// TIA Portal V15.1 export
// export: Created 2024-06-21T08:41:07.9526464Z, ExportSetting WithDefaults, DisplayName Totally Integrated Automation Portal, DisplayVersion V15.1 Update 5, DisplayName TIA Portal Openness, DisplayVersion V15.1 Update 5, DisplayName SINAMICS Startdrive Advanced, DisplayVersion V15.1, DisplayName G130, G150, S120, S150, SINAMICS MV, S210, DisplayVersion V15.1, DisplayName G110M, G120, G120C, G120D, G120P, DisplayVersion V15.1, DisplayName STEP 7 Professional, DisplayVersion V15.1 Update 5, DisplayName STEP 7 Safety, DisplayVersion V15.1, DisplayName WinCC Professional, DisplayVersion V15.1 Update 5, DisplayName SIMATIC Visualization Architect, DisplayVersion V15.1
FUNCTION_BLOCK "LGBInfeedOutfeed"   // FB6694, FBD
TITLE = LGBInfeedOutfeed
{ S7_Optimized_Access := 'TRUE' }
VERSION : 0.1
// stored: AutoNumber false, IsIECCheckEnabled false, IsRetainMemResEnabled false, MemoryReserve 100, SetENOAutomatically False, UDAEnableTagReadback false
   VAR_INPUT
      I_SelSwInfeed { ExternalAccessible := 'False'; ExternalVisible := 'False'; ExternalWritable := 'False'} : Bool;   // Selection switch Infeed selected
      I_SelSwOutfeed { ExternalAccessible := 'False'; ExternalVisible := 'False'; ExternalWritable := 'False'} : Bool;   // Selection switch Outfeed selected
      I_PBAcknowledge { ExternalAccessible := 'False'; ExternalVisible := 'False'; ExternalWritable := 'False'} : Bool;   // Pushbutton Acknowledge
      I_Pedal { ExternalAccessible := 'False'; ExternalVisible := 'False'; ExternalWritable := 'False'} : Bool;   // Pedal
      I_StopDet { ExternalAccessible := 'False'; ExternalVisible := 'False'; ExternalWritable := 'False'} : Bool;   // Stop detection roller during infeed
      I_ExtOutfeedReq { ExternalAccessible := 'False'; ExternalVisible := 'False'; ExternalWritable := 'False'} : Bool;   // External Outfeed request
      I_TrfOutRdyRcv { ExternalAccessible := 'False'; ExternalVisible := 'False'; ExternalWritable := 'False'} : Bool;   // Ready to Receive: Signal from next object
      I_TrfOutArrived { ExternalAccessible := 'False'; ExternalVisible := 'False'; ExternalWritable := 'False'} : Bool;   // Body Arrived: Signal from next object
      I_TrfInRdyDlv { ExternalAccessible := 'False'; ExternalVisible := 'False'; ExternalWritable := 'False'} : Bool;   // Ready to deliver: Signal from previous object
      I_TrfInTM { ExternalAccessible := 'False'; ExternalVisible := 'False'; ExternalWritable := 'False'} : Bool;   // Transfer busy signal from previous equipement
      C_TimeNotStopDet { ExternalAccessible := 'False'; ExternalVisible := 'False'; ExternalWritable := 'False'} : DInt;   // Time value for handshake signal "Arrived" by Infeed
   END_VAR
   VAR_OUTPUT
      O_TrfOutRdyDlv { ExternalAccessible := 'False'; ExternalVisible := 'False'; ExternalWritable := 'False'} : Bool;   // Ready to Deliver: Signal to next object
      O_TrfOutTM { ExternalAccessible := 'False'; ExternalVisible := 'False'; ExternalWritable := 'False'} : Bool;   // Transfer: Signal to next object
      O_TrfInRdyRcv { ExternalAccessible := 'False'; ExternalVisible := 'False'; ExternalWritable := 'False'} : Bool;   // Ready to Receive: Signal to previous object
      O_TrfInArrived { ExternalAccessible := 'False'; ExternalVisible := 'False'; ExternalWritable := 'False'} : Bool;   // Body Arrived: Signal to previous object
      O_ReqInfeed { ExternalAccessible := 'False'; ExternalVisible := 'False'; ExternalWritable := 'False'} : Bool;   // Infeed request / Led Infeed/Outfeed
      O_ReqOutfeed { ExternalAccessible := 'False'; ExternalVisible := 'False'; ExternalWritable := 'False'} : Bool;   // Outfeed request / Led Infeed/Outfeed
      O_LedInfeedOutfeed { ExternalAccessible := 'False'; ExternalVisible := 'False'; ExternalWritable := 'False'} : Bool;   // Led Infeed/Outfeed
      O_LedAcknowledge { ExternalAccessible := 'False'; ExternalVisible := 'False'; ExternalWritable := 'False'} : Bool;   // Led Acknowledge
      O_AlarmABCondition { ExternalAccessible := 'False'; ExternalVisible := 'False'; ExternalWritable := 'False'} : Bool;   // Alarm AB Condition
      O_AlarmA { ExternalAccessible := 'False'; ExternalVisible := 'False'; ExternalWritable := 'False'} : Bool;   // Alarm A
      O_AlarmB { ExternalAccessible := 'False'; ExternalVisible := 'False'; ExternalWritable := 'False'} : Bool;   // Alarm B
      O_AlarmC { ExternalAccessible := 'False'; ExternalVisible := 'False'; ExternalWritable := 'False'} : Bool;   // Alarm C
      O_AlarmD { ExternalAccessible := 'False'; ExternalVisible := 'False'; ExternalWritable := 'False'} : Bool;   // Alarm D
      H_AlarmDWord { ExternalAccessible := 'False'; ExternalVisible := 'False'; ExternalWritable := 'False'} : DWord;   // HMI Animation
   END_VAR
   VAR_IN_OUT
      IO_Modes : "Modes";   // Modes
      H_HMI : "H_HMI";   // Animation
      H_GBInfeedOutfeed : "H_GBInfeedOutfeed";   // Animation
   END_VAR
   VAR
      TrfOutRdyDlv { ExternalAccessible := 'False'; ExternalVisible := 'False'; ExternalWritable := 'False'} : Bool;   // Ready to Deliver: Signal to next object
      TrfOutTM { ExternalAccessible := 'False'; ExternalVisible := 'False'; ExternalWritable := 'False'} : Bool;   // Transfer: Signal to next object
      TrfInRdyRcv { ExternalAccessible := 'False'; ExternalVisible := 'False'; ExternalWritable := 'False'} : Bool;   // Ready to Receive: Signal to previous object
      TrfInArrived { ExternalAccessible := 'False'; ExternalVisible := 'False'; ExternalWritable := 'False'} : Bool;   // Body Arrived: Signal to previous object
      InfeedSel { ExternalAccessible := 'False'; ExternalVisible := 'False'; ExternalWritable := 'False'} : Bool;   // Infeed selected
      OutfeedSel { ExternalAccessible := 'False'; ExternalVisible := 'False'; ExternalWritable := 'False'} : Bool;   // Outfeed selected
      NotStopDetDelayed { ExternalAccessible := 'False'; ExternalVisible := 'False'; ExternalWritable := 'False'} : Bool;   // Not Stop detection delayted
      LedFeedInFeedOut { ExternalAccessible := 'False'; ExternalVisible := 'False'; ExternalWritable := 'False'} : Bool;   // Led Infeed/Outfeed
      LedAcknowledge { ExternalAccessible := 'False'; ExternalVisible := 'False'; ExternalWritable := 'False'} : Bool;   // Led Acknowledge
      ActNotStopDetDelayed { ExternalAccessible := 'False'; ExternalVisible := 'False'; ExternalWritable := 'False'} : DInt;   // Actual time Not Stop detection delayted
      AlarmA { ExternalAccessible := 'False'; ExternalVisible := 'False'; ExternalWritable := 'False'} : Bool;   // Alarm A
      AlarmB { ExternalAccessible := 'False'; ExternalVisible := 'False'; ExternalWritable := 'False'} : Bool;   // Alarm B
      AlarmC { ExternalAccessible := 'False'; ExternalVisible := 'False'; ExternalWritable := 'False'} : Bool;   // Alarm C
      AlarmD { ExternalAccessible := 'False'; ExternalVisible := 'False'; ExternalWritable := 'False'} : Bool;   // Alarm D
      AlarmABCondition { ExternalAccessible := 'False'; ExternalVisible := 'False'; ExternalWritable := 'False'} : Bool;   // Alarm AB Condition
      TimerNotStopDetDelayed { ExternalAccessible := 'False'; ExternalVisible := 'False'; ExternalWritable := 'False'} : "LTimer";   // FB
   END_VAR
   VAR_TEMP   // added for the SCL form of the ladder/FBD networks
      _w1 : Bool;
   END_VAR
BEGIN

REGION Network 1: **** 4.3 - Machine status - Operator selections **** Infeed selected
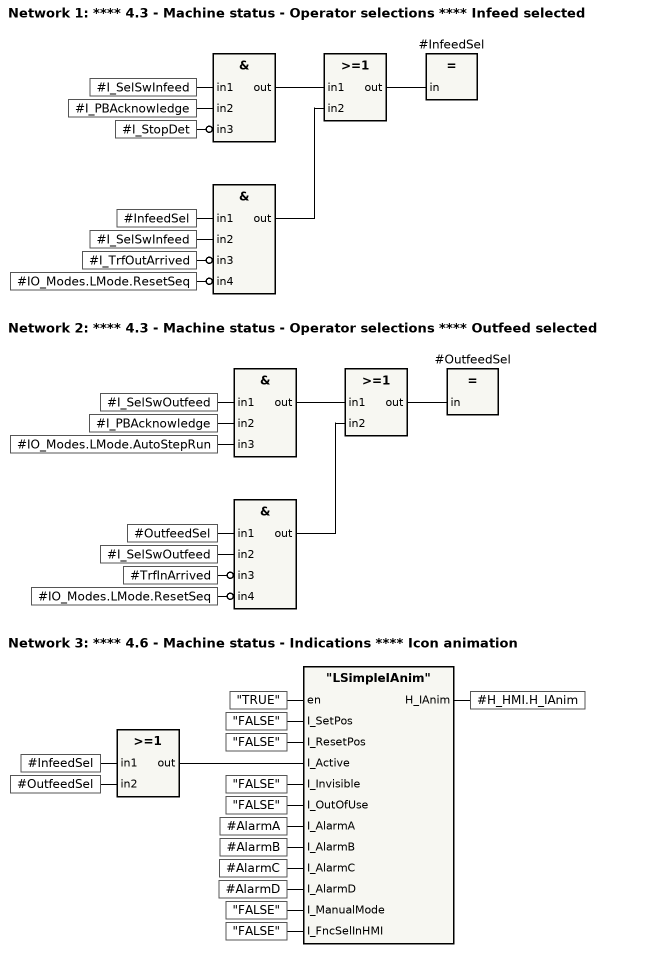
   #InfeedSel := (#I_SelSwInfeed AND #I_PBAcknowledge AND NOT #I_StopDet) OR (#InfeedSel AND #I_SelSwInfeed AND NOT #I_TrfOutArrived AND NOT #IO_Modes.LMode.ResetSeq);
END_REGION

REGION Network 2: **** 4.3 - Machine status - Operator selections **** Outfeed selected
   #OutfeedSel := (#I_SelSwOutfeed AND #I_PBAcknowledge AND #IO_Modes.LMode.AutoStepRun) OR (#OutfeedSel AND #I_SelSwOutfeed AND NOT #TrfInArrived AND NOT #IO_Modes.LMode.ResetSeq);
END_REGION

REGION Network 3: **** 4.6 - Machine status - Indications **** Icon animation
   // Icon animation
   IF "TRUE" THEN
       "LSimpleIAnim"(I_SetPos := "FALSE",
                      I_ResetPos := "FALSE",
                      I_Active := #InfeedSel OR #OutfeedSel,
                      I_Invisible := "FALSE",
                      I_OutOfUse := "FALSE",
                      I_AlarmA := #AlarmA,
                      I_AlarmB := #AlarmB,
                      I_AlarmC := #AlarmC,
                      I_AlarmD := #AlarmD,
                      I_ManualMode := "FALSE",
                      I_FncSelInHMI := "FALSE",
                      H_IAnim => #H_HMI.H_IAnim);
   END_IF;
END_REGION

REGION Network 4: **** 4.6 - Machine status - Indications **** Animation
   // Animation
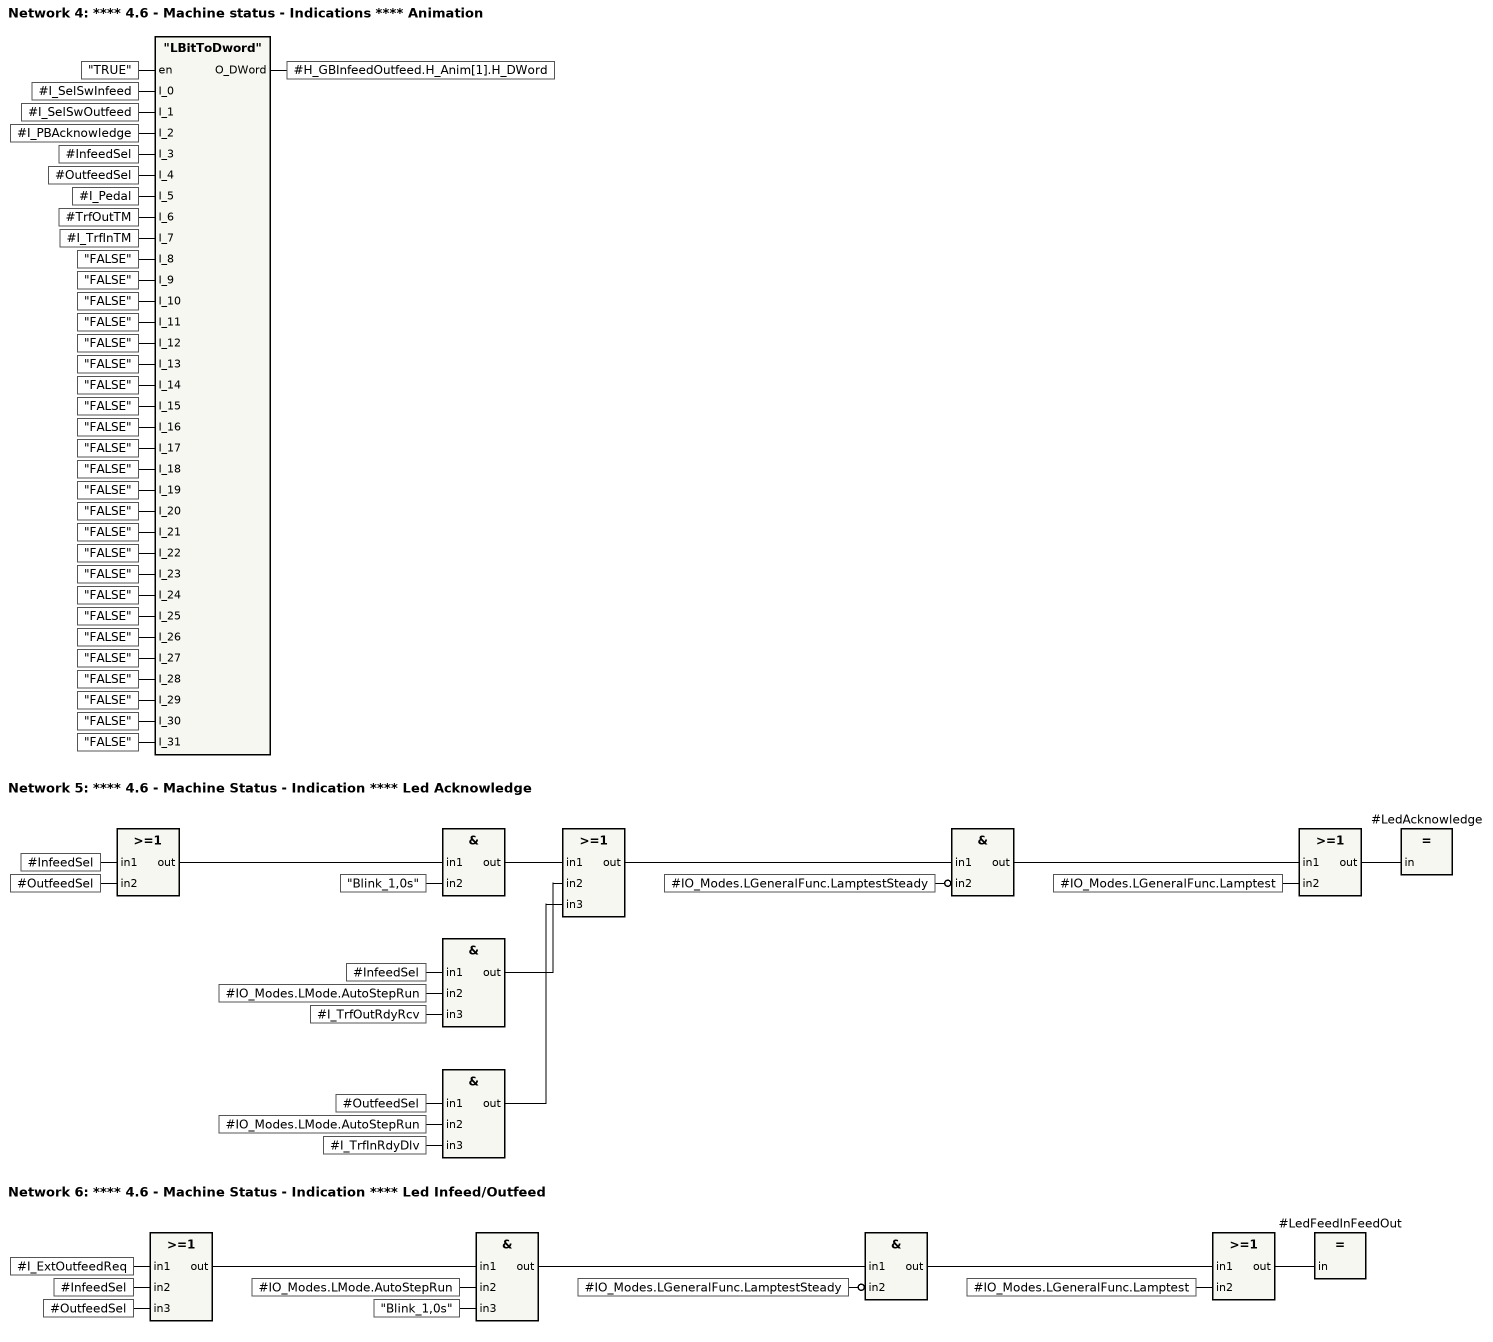
   IF "TRUE" THEN
       "LBitToDword"(I_0 := #I_SelSwInfeed,
                     I_1 := #I_SelSwOutfeed,
                     I_2 := #I_PBAcknowledge,
                     I_3 := #InfeedSel,
                     I_4 := #OutfeedSel,
                     I_5 := #I_Pedal,
                     I_6 := #TrfOutTM,
                     I_7 := #I_TrfInTM,
                     I_8 := "FALSE",
                     I_9 := "FALSE",
                     I_10 := "FALSE",
                     I_11 := "FALSE",
                     I_12 := "FALSE",
                     I_13 := "FALSE",
                     I_14 := "FALSE",
                     I_15 := "FALSE",
                     I_16 := "FALSE",
                     I_17 := "FALSE",
                     I_18 := "FALSE",
                     I_19 := "FALSE",
                     I_20 := "FALSE",
                     I_21 := "FALSE",
                     I_22 := "FALSE",
                     I_23 := "FALSE",
                     I_24 := "FALSE",
                     I_25 := "FALSE",
                     I_26 := "FALSE",
                     I_27 := "FALSE",
                     I_28 := "FALSE",
                     I_29 := "FALSE",
                     I_30 := "FALSE",
                     I_31 := "FALSE",
                     O_DWord => #H_GBInfeedOutfeed.H_Anim[1].H_DWord);
   END_IF;
END_REGION

REGION Network 5: **** 4.6 - Machine Status - Indication **** Led Acknowledge
   #LedAcknowledge := ((((#InfeedSel OR #OutfeedSel) AND "Blink_1,0s") OR (#InfeedSel AND #IO_Modes.LMode.AutoStepRun AND #I_TrfOutRdyRcv) OR (#OutfeedSel AND #IO_Modes.LMode.AutoStepRun AND #I_TrfInRdyDlv)) AND NOT #IO_Modes.LGeneralFunc.LamptestSteady) OR #IO_Modes.LGeneralFunc.Lamptest;
END_REGION

REGION Network 6: **** 4.6 - Machine Status - Indication **** Led Infeed/Outfeed
   #LedFeedInFeedOut := ((#I_ExtOutfeedReq OR #InfeedSel OR #OutfeedSel) AND #IO_Modes.LMode.AutoStepRun AND "Blink_1,0s" AND NOT #IO_Modes.LGeneralFunc.LamptestSteady) OR #IO_Modes.LGeneralFunc.Lamptest;
END_REGION

REGION Network 7: **** 5.2 - Equations - Flow Equation **** Timer Not StopDet Delayed
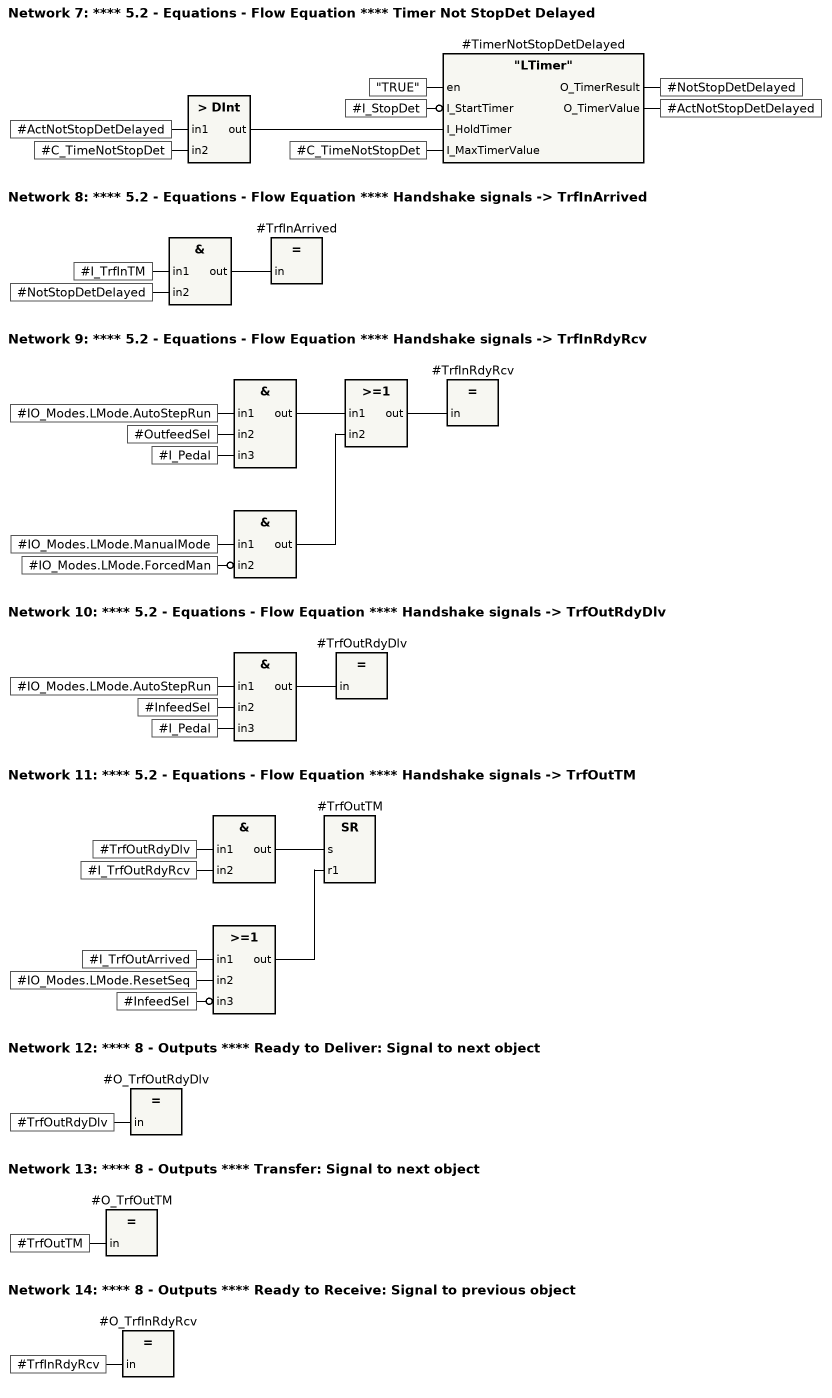
   IF "TRUE" THEN
       #TimerNotStopDetDelayed(I_StartTimer := NOT #I_StopDet,   // "LTimer"
                               I_HoldTimer := #ActNotStopDetDelayed > #C_TimeNotStopDet,
                               I_MaxTimerValue := #C_TimeNotStopDet,
                               O_TimerResult => #NotStopDetDelayed,
                               O_TimerValue => #ActNotStopDetDelayed);
   END_IF;
END_REGION

REGION Network 8: **** 5.2 - Equations - Flow Equation **** Handshake signals -> TrfInArrived
   #TrfInArrived := #I_TrfInTM AND #NotStopDetDelayed;
END_REGION

REGION Network 9: **** 5.2 - Equations - Flow Equation **** Handshake signals -> TrfInRdyRcv
   #TrfInRdyRcv := (#IO_Modes.LMode.AutoStepRun AND #OutfeedSel AND #I_Pedal) OR (#IO_Modes.LMode.ManualMode AND NOT #IO_Modes.LMode.ForcedMan);
END_REGION

REGION Network 10: **** 5.2 - Equations - Flow Equation **** Handshake signals -> TrfOutRdyDlv
   #TrfOutRdyDlv := #IO_Modes.LMode.AutoStepRun AND #InfeedSel AND #I_Pedal;
END_REGION

REGION Network 11: **** 5.2 - Equations - Flow Equation **** Handshake signals -> TrfOutTM
   IF #TrfOutRdyDlv AND #I_TrfOutRdyRcv THEN
       #TrfOutTM := TRUE;   // SR flip-flop
   END_IF;
   IF #I_TrfOutArrived OR #IO_Modes.LMode.ResetSeq OR NOT #InfeedSel THEN #TrfOutTM := FALSE; END_IF;
END_REGION

REGION Network 12: **** 8 - Outputs **** Ready to Deliver: Signal to next object
   #O_TrfOutRdyDlv := #TrfOutRdyDlv;
END_REGION

REGION Network 13: **** 8 - Outputs **** Transfer: Signal to next object
   #O_TrfOutTM := #TrfOutTM;
END_REGION

REGION Network 14: **** 8 - Outputs **** Ready to Receive: Signal to previous object
   #O_TrfInRdyRcv := #TrfInRdyRcv;
END_REGION

REGION Network 15: **** 8 - Outputs **** Body Arrived: Signal to previous object
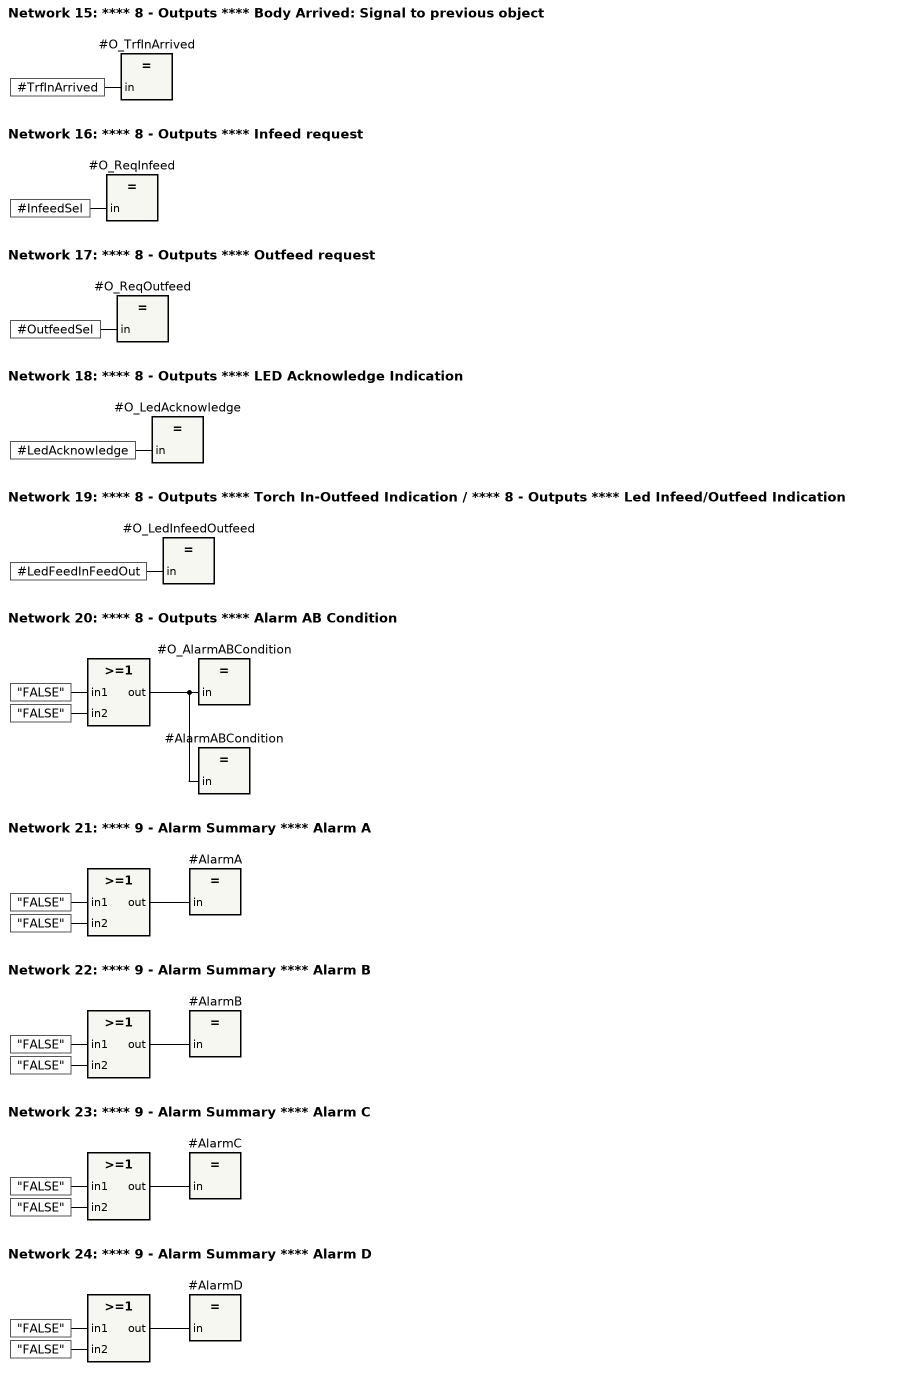
   #O_TrfInArrived := #TrfInArrived;
END_REGION

REGION Network 16: **** 8 - Outputs **** Infeed request
   #O_ReqInfeed := #InfeedSel;
END_REGION

REGION Network 17: **** 8 - Outputs **** Outfeed request
   #O_ReqOutfeed := #OutfeedSel;
END_REGION

REGION Network 18: **** 8 - Outputs **** LED Acknowledge Indication
   #O_LedAcknowledge := #LedAcknowledge;
END_REGION

REGION Network 19: **** 8 - Outputs **** Torch In-Outfeed Indication / **** 8 - Outputs **** Led Infeed/Outfeed Indication
   #O_LedInfeedOutfeed := #LedFeedInFeedOut;
END_REGION

REGION Network 20: **** 8 - Outputs **** Alarm AB Condition
   // Alarm AB Condition
   #O_AlarmABCondition := "FALSE" OR "FALSE";
   #AlarmABCondition := #O_AlarmABCondition;
END_REGION

REGION Network 21: **** 9 - Alarm Summary **** Alarm A
   // Alarm A
   #AlarmA := "FALSE" OR "FALSE";
END_REGION

REGION Network 22: **** 9 - Alarm Summary **** Alarm B
   // Alarm B
   #AlarmB := "FALSE" OR "FALSE";
END_REGION

REGION Network 23: **** 9 - Alarm Summary **** Alarm C
   // Alarm C
   #AlarmC := "FALSE" OR "FALSE";
END_REGION

REGION Network 24: **** 9 - Alarm Summary **** Alarm D
   // Alarm D
   #AlarmD := "FALSE" OR "FALSE";
END_REGION

REGION Network 25: **** 9 - Alarm Summary **** Alarms To Alarm UDT Alarms To Alarm UDT Get Name
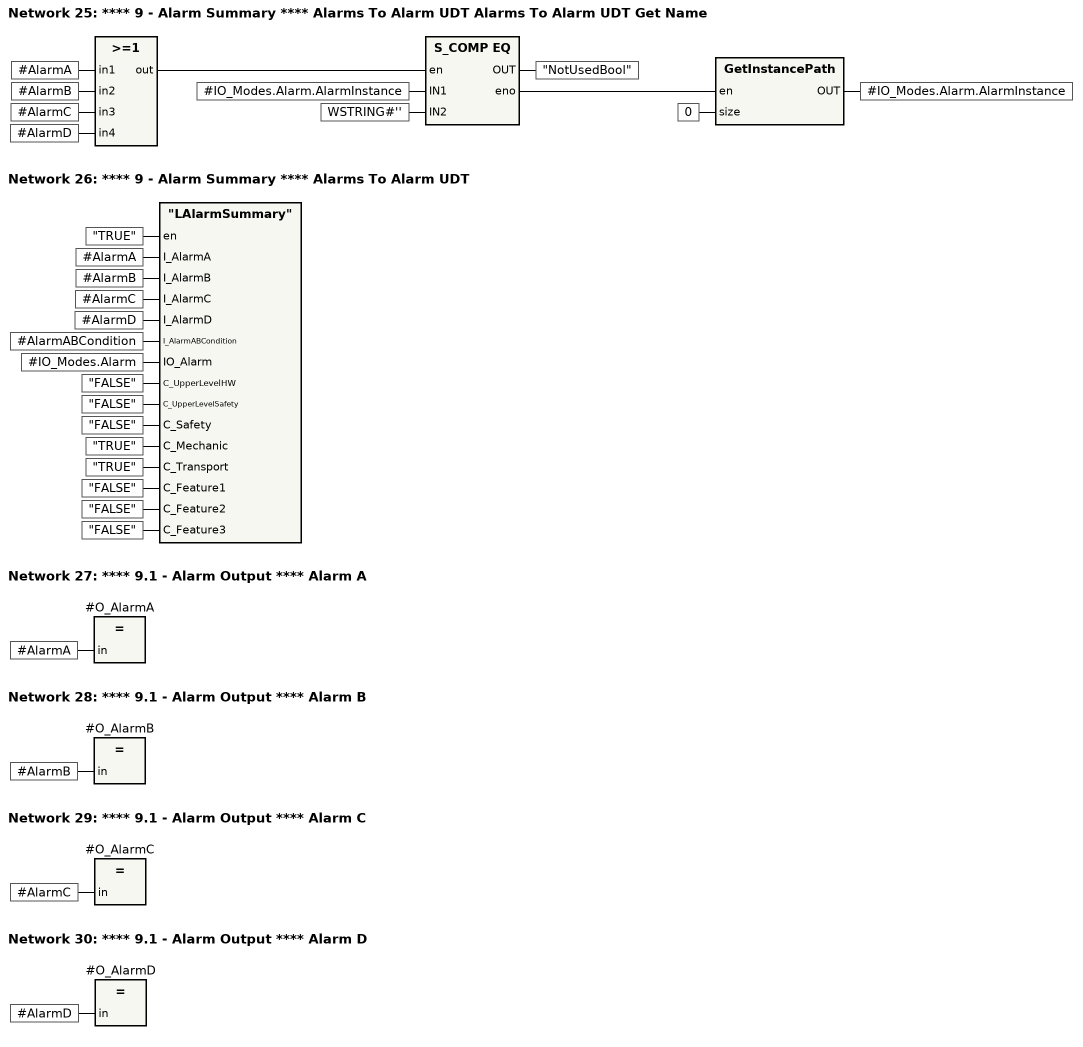
   S_COMP(EN := #AlarmA OR #AlarmB OR #AlarmC OR #AlarmD,
          IN1 := #IO_Modes.Alarm.AlarmInstance,
          IN2 := WSTRING#'',
          OUT => "NotUsedBool",
          ENO => #_w1);
   IF #_w1 THEN GetInstancePath(size := 0, OUT => #IO_Modes.Alarm.AlarmInstance); END_IF;
END_REGION

REGION Network 26: **** 9 - Alarm Summary **** Alarms To Alarm UDT
   IF "TRUE" THEN
       "LAlarmSummary"(I_AlarmA := #AlarmA,
                       I_AlarmB := #AlarmB,
                       I_AlarmC := #AlarmC,
                       I_AlarmD := #AlarmD,
                       I_AlarmABCondition := #AlarmABCondition,
                       IO_Alarm := #IO_Modes.Alarm,
                       C_UpperLevelHW := "FALSE",
                       C_UpperLevelSafety := "FALSE",
                       C_Safety := "FALSE",
                       C_Mechanic := "TRUE",
                       C_Transport := "TRUE",
                       C_Feature1 := "FALSE",
                       C_Feature2 := "FALSE",
                       C_Feature3 := "FALSE");
   END_IF;
END_REGION

REGION Network 27: **** 9.1 - Alarm Output **** Alarm A
   // Alarm A
   #O_AlarmA := #AlarmA;
END_REGION

REGION Network 28: **** 9.1 - Alarm Output **** Alarm B
   // Alarm B
   #O_AlarmB := #AlarmB;
END_REGION

REGION Network 29: **** 9.1 - Alarm Output **** Alarm C
   // Alarm C
   #O_AlarmC := #AlarmC;
END_REGION

REGION Network 30: **** 9.1 - Alarm Output **** Alarm D
   // Alarm D
   #O_AlarmD := #AlarmD;
END_REGION

REGION Network 31: **** 9.2 - Alarm DWord**** Alarm To DWord
   // Alarm To Word
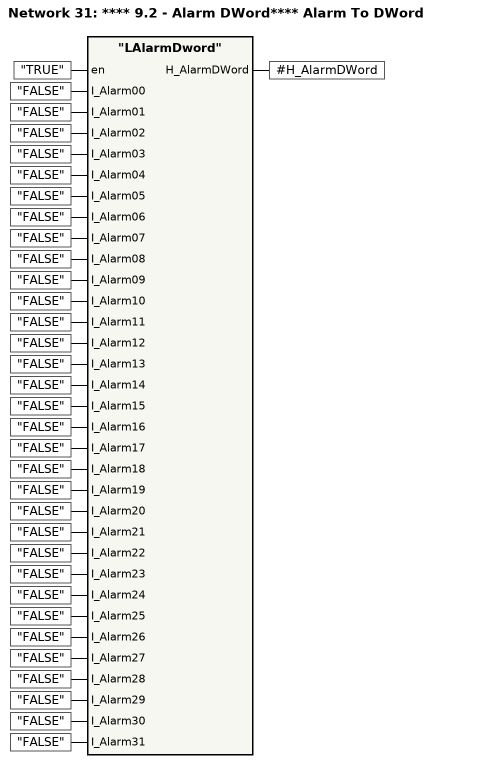
   IF "TRUE" THEN
       "LAlarmDword"(I_Alarm00 := "FALSE",
                     I_Alarm01 := "FALSE",
                     I_Alarm02 := "FALSE",
                     I_Alarm03 := "FALSE",
                     I_Alarm04 := "FALSE",
                     I_Alarm05 := "FALSE",
                     I_Alarm06 := "FALSE",
                     I_Alarm07 := "FALSE",
                     I_Alarm08 := "FALSE",
                     I_Alarm09 := "FALSE",
                     I_Alarm10 := "FALSE",
                     I_Alarm11 := "FALSE",
                     I_Alarm12 := "FALSE",
                     I_Alarm13 := "FALSE",
                     I_Alarm14 := "FALSE",
                     I_Alarm15 := "FALSE",
                     I_Alarm16 := "FALSE",
                     I_Alarm17 := "FALSE",
                     I_Alarm18 := "FALSE",
                     I_Alarm19 := "FALSE",
                     I_Alarm20 := "FALSE",
                     I_Alarm21 := "FALSE",
                     I_Alarm22 := "FALSE",
                     I_Alarm23 := "FALSE",
                     I_Alarm24 := "FALSE",
                     I_Alarm25 := "FALSE",
                     I_Alarm26 := "FALSE",
                     I_Alarm27 := "FALSE",
                     I_Alarm28 := "FALSE",
                     I_Alarm29 := "FALSE",
                     I_Alarm30 := "FALSE",
                     I_Alarm31 := "FALSE",
                     H_AlarmDWord => #H_AlarmDWord);
   END_IF;
END_REGION
END_FUNCTION_BLOCK
